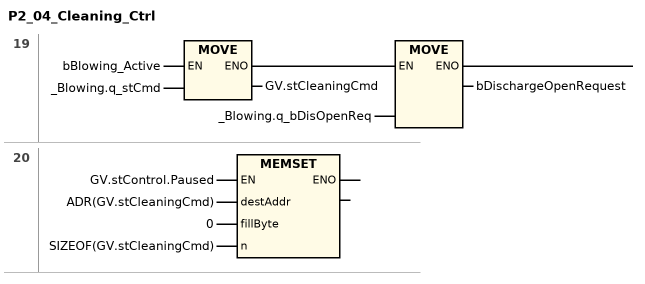
// NETWORK 19
_w4 := bBlowing_Active;
IF _w4 THEN GV.stCleaningCmd := _Blowing.q_stCmd; END_IF
IF _w4 THEN bDischargeOpenRequest := _Blowing.q_bDisOpenReq; END_IF

// NETWORK 20
IF GV.stControl.Paused THEN
    MEMSET(destAddr := ADR(GV.stCleaningCmd), fillByte := 0, n := SIZEOF(GV.stCleaningCmd));
END_IF

END_PROGRAM

// ---- POUs/2. Process/P2_05_Process_Ctrl.TcPOU
PROGRAM P2_05_Process_Ctrl
VAR
	bWaitAferBatchClose			:BOOL;
	tonWaitAfterBatchClose		:TON;
	tonMixerDelayStopped: TON;
END_VAR
VAR // added by the converter: edge detectors and wires of the graphical bodies
    _w1, _w2, _w3 : BOOL;
    _rt1 : R_TRIG;
END_VAR

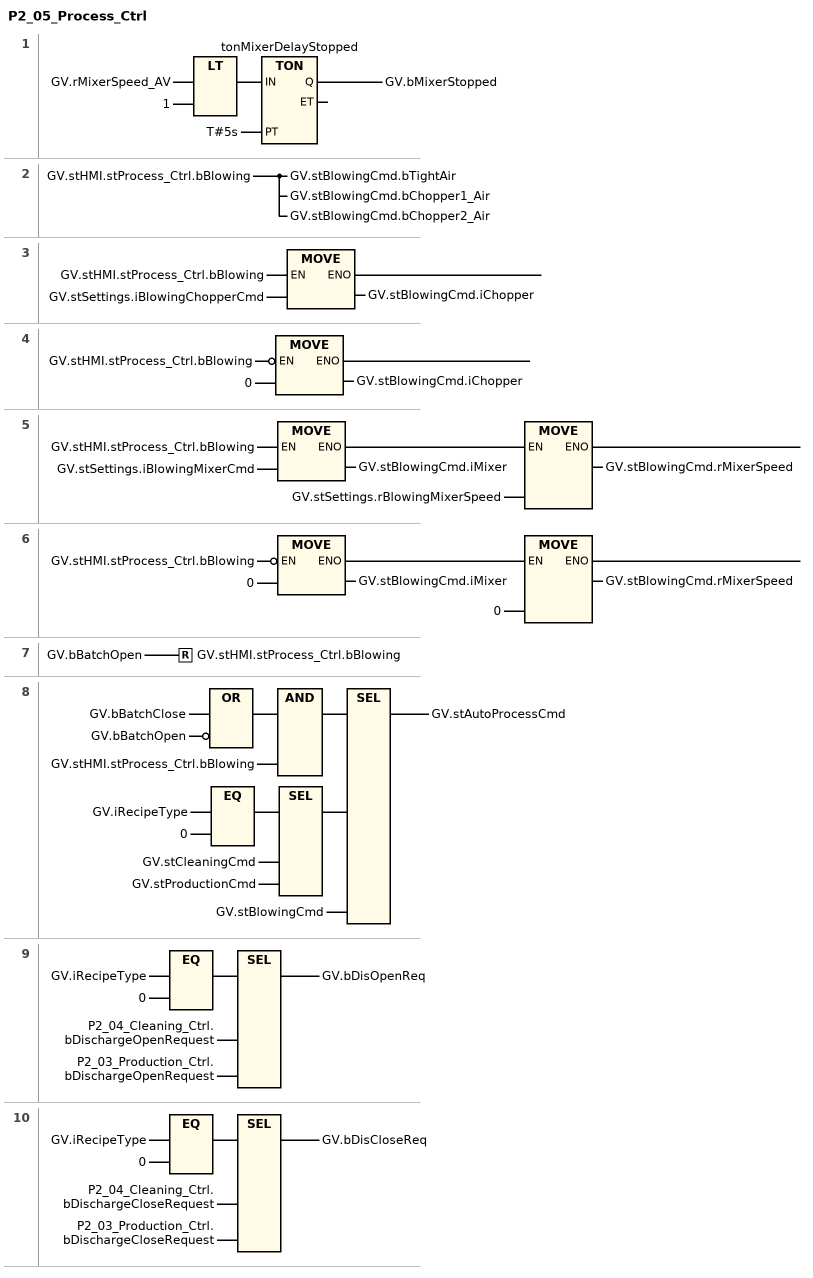
// NETWORK 1
tonMixerDelayStopped(IN := GV.rMixerSpeed_AV < 1, PT := T#5s); // TON
GV.bMixerStopped := tonMixerDelayStopped.Q;

// NETWORK 2
_w1 := GV.stHMI.stProcess_Ctrl.bBlowing;
GV.stBlowingCmd.bTightAir := _w1;
GV.stBlowingCmd.bChopper1_Air := _w1;
GV.stBlowingCmd.bChopper2_Air := _w1;

// NETWORK 3
IF GV.stHMI.stProcess_Ctrl.bBlowing THEN GV.stBlowingCmd.iChopper := GV.stSettings.iBlowingChopperCmd; END_IF

// NETWORK 4
IF NOT GV.stHMI.stProcess_Ctrl.bBlowing THEN GV.stBlowingCmd.iChopper := 0; END_IF

// NETWORK 5
_w2 := GV.stHMI.stProcess_Ctrl.bBlowing;
IF _w2 THEN GV.stBlowingCmd.iMixer := GV.stSettings.iBlowingMixerCmd; END_IF
IF _w2 THEN GV.stBlowingCmd.rMixerSpeed := GV.stSettings.rBlowingMixerSpeed; END_IF

// NETWORK 6
_w3 := NOT GV.stHMI.stProcess_Ctrl.bBlowing;
IF _w3 THEN GV.stBlowingCmd.iMixer := 0; END_IF
IF _w3 THEN GV.stBlowingCmd.rMixerSpeed := 0; END_IF

// NETWORK 7
GV.stHMI.stProcess_Ctrl.bBlowing R= GV.bBatchOpen;

// NETWORK 8
GV.stAutoProcessCmd := SEL((GV.bBatchClose OR NOT GV.bBatchOpen) AND GV.stHMI.stProcess_Ctrl.bBlowing, SEL(GV.iRecipeType = 0, GV.stCleaningCmd, GV.stProductionCmd), GV.stBlowingCmd);

// NETWORK 9
GV.bDisOpenReq := SEL(GV.iRecipeType = 0, P2_04_Cleaning_Ctrl.bDischargeOpenRequest, P2_03_Production_Ctrl.bDischargeOpenRequest);

// NETWORK 10
GV.bDisCloseReq := SEL(GV.iRecipeType = 0, P2_04_Cleaning_Ctrl.bDischargeCloseRequest, P2_03_Production_Ctrl.bDischargeCloseRequest);

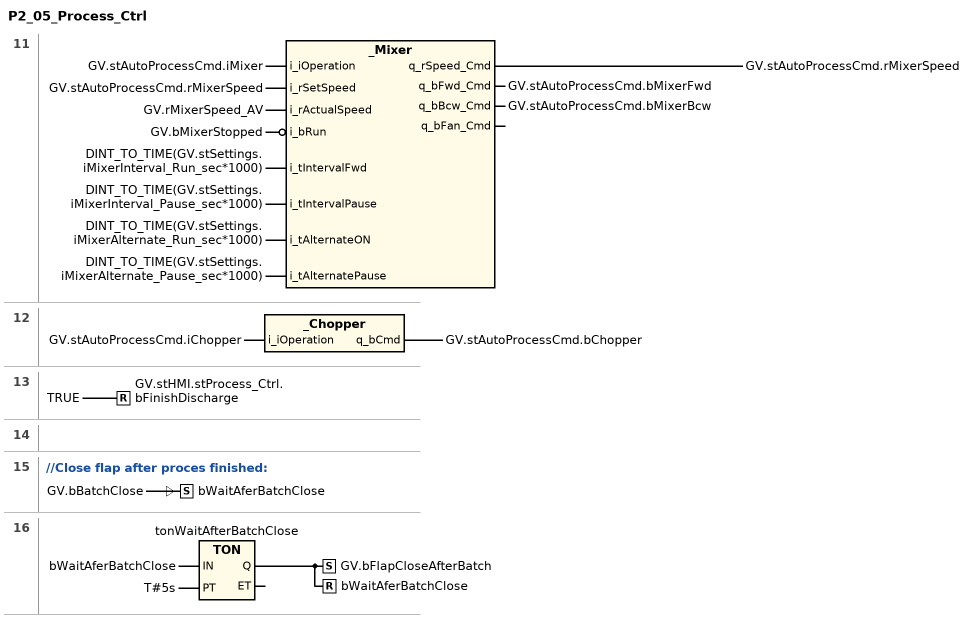
// NETWORK 11
_Mixer(i_iOperation := GV.stAutoProcessCmd.iMixer, i_rSetSpeed := GV.stAutoProcessCmd.rMixerSpeed, i_rActualSpeed := GV.rMixerSpeed_AV, i_bRun := NOT GV.bMixerStopped, i_tIntervalFwd := DINT_TO_TIME(GV.stSettings.iMixerInterval_Run_sec*1000), i_tIntervalPause := DINT_TO_TIME(GV.stSettings.iMixerInterval_Pause_sec*1000), i_tAlternateON := DINT_TO_TIME(GV.stSettings.iMixerAlternate_Run_sec*1000), i_tAlternatePause := DINT_TO_TIME(GV.stSettings.iMixerAlternate_Pause_sec*1000), q_bFwd_Cmd => GV.stAutoProcessCmd.bMixerFwd, q_bBcw_Cmd => GV.stAutoProcessCmd.bMixerBcw);
GV.stAutoProcessCmd.rMixerSpeed := _Mixer.q_rSpeed_Cmd;

// NETWORK 12
_Chopper(i_iOperation := GV.stAutoProcessCmd.iChopper);
GV.stAutoProcessCmd.bChopper := _Chopper.q_bCmd;

// NETWORK 13
GV.stHMI.stProcess_Ctrl.bFinishDischarge R= TRUE;

// NETWORK 14

// NETWORK 15
// label: //Close flap after proces finished
_rt1(CLK := GV.bBatchClose);
bWaitAferBatchClose S= _rt1.Q;

// NETWORK 16
tonWaitAfterBatchClose(IN := bWaitAferBatchClose, PT := T#5s); // TON
GV.bFlapCloseAfterBatch S= tonWaitAfterBatchClose.Q;
bWaitAferBatchClose R= tonWaitAfterBatchClose.Q;

END_PROGRAM

// ---- POUs/2. Process/_Chopper.TcPOU
PROGRAM _Chopper
VAR_INPUT
	i_iOperation			:INT;
END_VAR

VAR
END_VAR

VAR_OUTPUT
	q_bCmd					:BOOL;
END_VAR

IF i_iOperation <> 0 THEN
	IF i_iOperation = 1 THEN
		q_bCmd:=TRUE;
	END_IF
ELSE
	q_bCmd:=FALSE;
END_IF

END_PROGRAM

// ---- POUs/3. Report/P3_00_MAIN.TcPOU
PROGRAM P3_00_MAIN
VAR
	tonDeleteDelay			:TON;
END_VAR

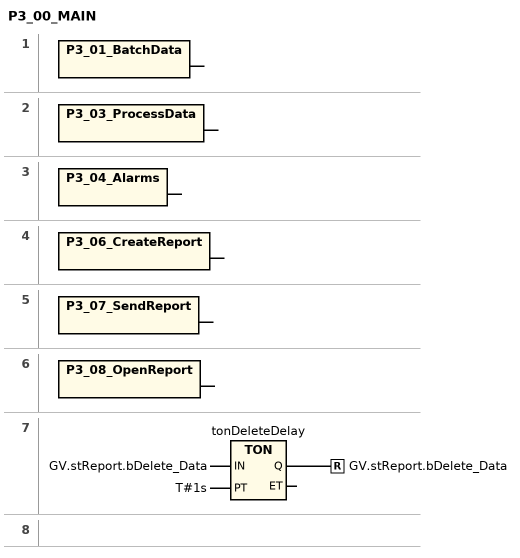
// NETWORK 1
P3_01_BatchData();

// NETWORK 2
P3_03_ProcessData();

// NETWORK 3
P3_04_Alarms();

// NETWORK 4
P3_06_CreateReport();

// NETWORK 5
P3_07_SendReport();

// NETWORK 6
P3_08_OpenReport();

// NETWORK 7
tonDeleteDelay(IN := GV.stReport.bDelete_Data, PT := T#1s); // TON
GV.stReport.bDelete_Data R= tonDeleteDelay.Q;

// NETWORK 8

END_PROGRAM

// ---- POUs/3. Report/P3_01_BatchData.TcPOU
PROGRAM P3_01_BatchData
VAR
	
	arrBatchParam				:ARRAY[0..19] OF STRING;
	arrBatchValue				:ARRAY[0..19] OF STRING;
	
	iNoParameters				:INT;
	
	stDBParam 					:ST_BatchData;	
	fbDBWrite					:FB_PLCDBWriteEvt(sNetId:=CONST.AMS_NETID, tTimeout:=DEFAULT_ADS_TIMEOUT);
	tableColumns				:ARRAY [0..2] OF STRING(50) := ['Batch', 'Parameter', 'Value'];
	arrParam					:ARRAY [0..2] OF ST_ExpParameter := [(sParaName := 'Batch', nParaSize := 101, eParaType := E_EXPPARAMETERTYPE.STRING_), 
																	(sParaName := 'Parameter', nParaSize := 101, eParaType := E_EXPPARAMETERTYPE.STRING_),
															 		(sParaName := 'Value', nParaSize := 101, eParaType := E_EXPPARAMETERTYPE.STRING_)];
															 
	fbDeleteTable    			:FB_PLCDBCmdEvt(sNetID:=CONST.AMS_NETID, tTimeout:=DEFAULT_ADS_TIMEOUT);	
	sDelete						:STRING;	
	bDelete						:BOOL;
															 
	bWrite						:BOOL;
	iWrite						:USINT;
	bStartWrite					:BOOL;
	
	sVersion					:STRING;
	
	iStepWrite					:INT;
	trigStartWrite				:R_TRIG;
	tonDelayWrite				:TON;
	
END_VAR
VAR PERSISTENT
	dtBatchOpen					:DT;
	dtBatchClose				:DT;
	
	ulBatchOpen					:ULINT;
	ulBatchClose				:ULINT;
END_VAR
VAR // added by the converter: edge detectors and wires of the graphical bodies
    _rt1, _rt2 : R_TRIG;
    _w1, _w2 : BOOL;
END_VAR

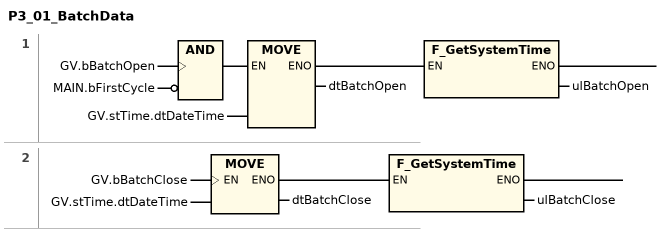
// NETWORK 1
_rt1(CLK := GV.bBatchOpen);
_w1 := _rt1.Q AND NOT MAIN.bFirstCycle;
IF _w1 THEN dtBatchOpen := GV.stTime.dtDateTime; END_IF
IF _w1 THEN ulBatchOpen := F_GetSystemTime(); END_IF

// NETWORK 2
_rt2(CLK := GV.bBatchClose);
_w2 := _rt2.Q;
IF _w2 THEN dtBatchClose := GV.stTime.dtDateTime; END_IF
IF _w2 THEN ulBatchClose := F_GetSystemTime(); END_IF

END_PROGRAM

// ---- POUs/3. Report/P3_03_ProcessData.TcPOU
PROGRAM P3_03_ProcessData
VAR
	stDBParam 					:ST_ProcessData;	

	fbDBWrite					:FB_PLCDBWriteEvt(sNetId:=CONST.AMS_NETID, tTimeout:=DEFAULT_ADS_TIMEOUT);
	tableColumns				:ARRAY [0..8] OF STRING(50) := ['Batch', 'DateTime', 'Value1', 'Value2', 'Value3', 'Value4', 'Value5', 'Value6', 'Value7'];
	arrParam					:ARRAY [0..8] OF ST_ExpParameter := [(sParaName := 'Batch', nParaSize := 101, eParaType := E_EXPPARAMETERTYPE.STRING_),
															 (sParaName := 'DateTime', nParaSize := 4, eParaType := E_EXPPARAMETERTYPE.DateTime), 
															 (sParaName := 'Value1', nParaSize := 101, eParaType := E_EXPPARAMETERTYPE.STRING_), 
															 (sParaName := 'Value2', nParaSize := 101, eParaType := E_EXPPARAMETERTYPE.STRING_), 
															 (sParaName := 'Value3', nParaSize := 101, eParaType := E_EXPPARAMETERTYPE.STRING_),
															 (sParaName := 'Value4', nParaSize := 101, eParaType := E_EXPPARAMETERTYPE.STRING_),
															 (sParaName := 'Value5', nParaSize := 101, eParaType := E_EXPPARAMETERTYPE.STRING_),
															 (sParaName := 'Value6', nParaSize := 101, eParaType := E_EXPPARAMETERTYPE.STRING_),
															 (sParaName := 'Value7', nParaSize := 101, eParaType := E_EXPPARAMETERTYPE.STRING_)];
		
	fbDeleteTable    			:FB_PLCDBCmdEvt(sNetID:=CONST.AMS_NETID, tTimeout:=DEFAULT_ADS_TIMEOUT);	
	sDelete						:STRING;	
	bDelete						:BOOL;
										 
	bWrite						:BOOL;	
	
	sChopper1Speed				:STRING;
	sChopper2Speed				:STRING;
END_VAR
VAR // added by the converter: edge detectors and wires of the graphical bodies
    _rt1, _rt2 : R_TRIG;
END_VAR

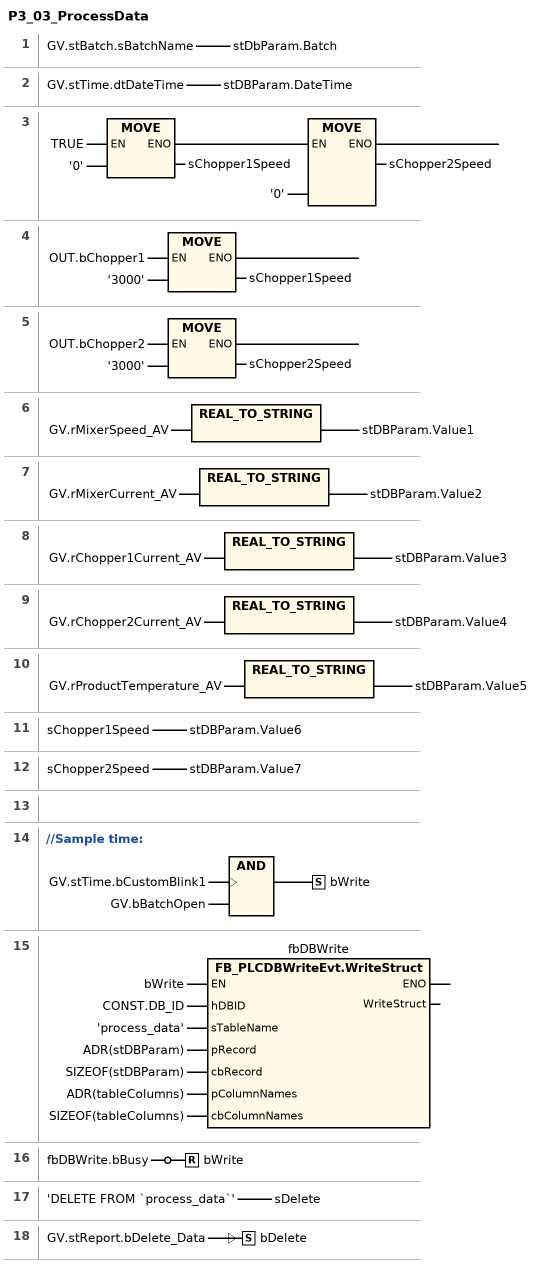
// NETWORK 1
stDbParam.Batch := GV.stBatch.sBatchName;

// NETWORK 2
stDBParam.DateTime := GV.stTime.dtDateTime;

// NETWORK 3
sChopper1Speed := '0';
sChopper2Speed := '0';

// NETWORK 4
IF OUT.bChopper1 THEN sChopper1Speed := '3000'; END_IF

// NETWORK 5
IF OUT.bChopper2 THEN sChopper2Speed := '3000'; END_IF

// NETWORK 6
stDBParam.Value1 := REAL_TO_STRING(GV.rMixerSpeed_AV);

// NETWORK 7
stDBParam.Value2 := REAL_TO_STRING(GV.rMixerCurrent_AV);

// NETWORK 8
stDBParam.Value3 := REAL_TO_STRING(GV.rChopper1Current_AV);

// NETWORK 9
stDBParam.Value4 := REAL_TO_STRING(GV.rChopper2Current_AV);

// NETWORK 10
stDBParam.Value5 := REAL_TO_STRING(GV.rProductTemperature_AV);

// NETWORK 11
stDBParam.Value6 := sChopper1Speed;

// NETWORK 12
stDBParam.Value7 := sChopper2Speed;

// NETWORK 13

// NETWORK 14
// label: //Sample time
_rt1(CLK := GV.stTime.bCustomBlink1);
bWrite S= _rt1.Q AND GV.bBatchOpen;

// NETWORK 15
IF bWrite THEN
    fbDBWrite.WriteStruct(
        hDBID := CONST.DB_ID,
        sTableName := 'process_data',
        pRecord := ADR(stDBParam),
        cbRecord := SIZEOF(stDBParam),
        pColumnNames := ADR(tableColumns),
        cbColumnNames := SIZEOF(tableColumns));
END_IF

// NETWORK 16
bWrite R= NOT fbDBWrite.bBusy;

// NETWORK 17
sDelete := 'DELETE FROM `process_data`';

// NETWORK 18
_rt2(CLK := GV.stReport.bDelete_Data);
bDelete S= _rt2.Q;

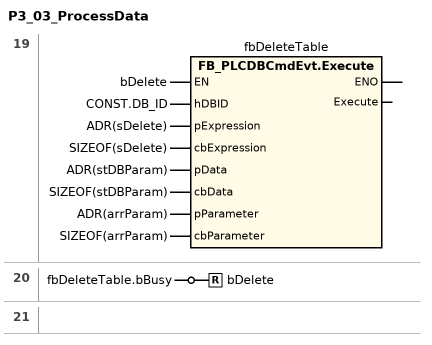
// NETWORK 19
IF bDelete THEN
    fbDeleteTable.Execute(
        hDBID := CONST.DB_ID,
        pExpression := ADR(sDelete),
        cbExpression := SIZEOF(sDelete),
        pData := ADR(stDBParam),
        cbData := SIZEOF(stDBParam),
        pParameter := ADR(arrParam),
        cbParameter := SIZEOF(arrParam));
END_IF

// NETWORK 20
bDelete R= NOT fbDeleteTable.bBusy;

// NETWORK 21

END_PROGRAM

// ---- POUs/3. Report/P3_04_Alarms.TcPOU
PROGRAM P3_04_Alarms
VAR 
	fbEventLogger		:FB_TcEventLogger;
	fbCsvExportSetting	:FB_TcEventCsvExportSettings;
	fbExportFilter		:FB_TcEventFilter;

	fbTrig				:R_TRIG;
	
	ulFilter1			:ULINT;
	ulFilter2			:ULINT;
	
	sPath				:STRING;
	
	
END_VAR

//Link here...

ulFilter1:=P3_01_BatchData.ulBatchOpen;
ulFilter2:=P3_01_BatchData.ulBatchClose;

fbTrig(CLK:=GV.stReport.bExport_Alarms);
IF GV.stReport.bExport_Alarms THEN
	IF fbTrig.Q THEN
		fbCsvExportSetting.Clear();
		fbCsvExportSetting.bWithHeader:=TRUE;
		fbCsvExportSetting.sDelimiter:=',';
		fbCsvExportSetting.AddFilter(fbExportFilter);
		fbExportFilter.Clear();
		fbExportFilter.IsAlarm().AND_OP().
		TimeRaised.GreaterThanOrEqualTo(ulFilter1).AND_OP().
		TimeRaised.LessThanOrEqualTo(ulFilter2).AND_OP().
		Source.Name.EqualTo('GV.stAlarm');
	END_IF
	
	sPath:=CONCAT(CONST.PROJECT_DIR,'Reports\1. Raw Data\AlarmLog.txt');
	
	IF fbEventLogger.ExportLoggedEvents(sPath,fbCsvExportSetting) THEN
		GV.stReport.bExport_Alarms:=FALSE;
	END_IF
END_IF

END_PROGRAM

// ---- POUs/3. Report/P3_08_OpenReport.TcPOU
PROGRAM P3_08_OpenReport
VAR
	sDateTime			:STRING;
	sYear				:STRING;
	sMonth				:STRING;
	sDay				:STRING;
	sHour				:STRING;
	sMinute				:STRING;
	sReportSuffix		:STRING;
END_VAR

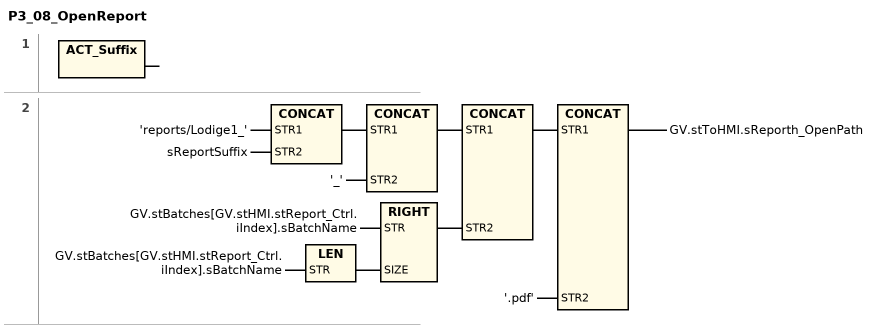
// NETWORK 1
ACT_Suffix();

// NETWORK 2
GV.stToHMI.sReporth_OpenPath := CONCAT(STR1 := CONCAT(STR1 := CONCAT(STR1 := CONCAT(STR1 := 'reports/Lodige1_', STR2 := sReportSuffix), STR2 := '_'), STR2 := RIGHT(STR := GV.stBatches[GV.stHMI.stReport_Ctrl.iIndex].sBatchName, SIZE := LEN(STR := GV.stBatches[GV.stHMI.stReport_Ctrl.iIndex].sBatchName))), STR2 := '.pdf');

ACTION ACT_Suffix:
sDateTime:=GV.stBatches[GV.stHMI.stReport_Ctrl.iIndex].sFinished;
sYear:=RIGHT(LEFT(sDateTime,10),2);
sMonth:=RIGHT(LEFT(sDateTime,5),2);
sDay:=LEFT(sDateTime,2);

sHour:=LEFT(RIGHT(sDateTime,8),2);
sMinute:=LEFT(RIGHT(sDateTime,5),2);

sReportSuffix:=CONCAT(sYear,sMonth);
sReportSuffix:=CONCAT(sReportSuffix,sDay);
sReportSuffix:=CONCAT(sReportSuffix,sHour);
sReportSuffix:=CONCAT(sReportSuffix,sMinute);
END_ACTION

END_PROGRAM

// ---- POUs/4. Audit Trail/P4_00_MAIN.TcPOU
PROGRAM P4_00_MAIN
VAR
END_VAR

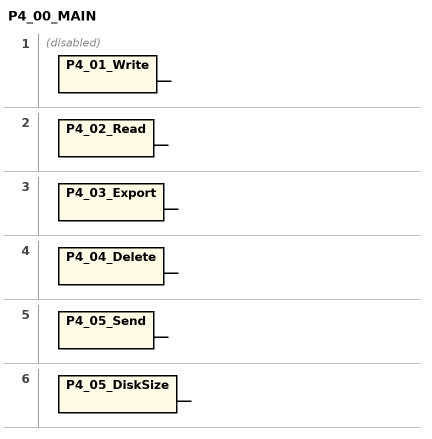
// NETWORK 1 (disabled)
// P4_01_Write();

// NETWORK 2
P4_02_Read();

// NETWORK 3
P4_03_Export();

// NETWORK 4
P4_04_Delete();

// NETWORK 5
P4_05_Send();

// NETWORK 6
P4_05_DiskSize();

END_PROGRAM

// ---- POUs/4. Audit Trail/P4_01_Write.TcPOU
PROGRAM P4_01_Write
VAR
	stDBParam 				:ST_AuditTrail;	
	tableColumns			:ARRAY [0..5] OF STRING(50) := ['DateTime', 'User', 'Event', 'Description', 'OldValue', 'NewValue'];	

	fbDBWrite				:FB_PLCDBWriteEvt(sNetId:=CONST.AMS_NETID, tTimeout:=DEFAULT_ADS_TIMEOUT);	
	bWrite					:BOOL;
	

	
	fbRecipeProdValue		:ARRAY[0..9] OF FB_WriteChange;
	fbRecipeProdStrings		:ARRAY[0..9] OF FB_WriteChange_STR;
	fbRecipeProdClick		:ARRAY[0..9] OF FB_WriteClick;
	bRecipeProdChange		:ARRAY[0..19] OF BOOL;
	
	fbRecipeCleanValue		:ARRAY[0..29] OF FB_WriteChange;
	fbRecipeCleanStrings	:ARRAY[0..29] OF FB_WriteChange_STR;
	fbRecipeCleanClick		:ARRAY[0..29] OF FB_WriteClick;
	bRecipeCleanChange		:ARRAY[0..39] OF BOOL;
	
	fbBatchProdValue		:ARRAY[0..9] OF FB_WriteChange;
	fbBatchProdStrings		:ARRAY[0..9] OF FB_WriteChange_STR;
	fbBatchProdClick		:ARRAY[0..9] OF FB_WriteClick;
	bBatchProdChange		:ARRAY[0..19] OF BOOL;
	
	fbBatchCleanValue		:ARRAY[0..29] OF FB_WriteChange;
	fbBatchCleanStrings		:ARRAY[0..29] OF FB_WriteChange_STR;
	fbBatchCleanClick		:ARRAY[0..29] OF FB_WriteClick;
	bBatchCleanChange		:ARRAY[0..39] OF BOOL;
	
	
	fbSettingsChange		:ARRAY[0..19] OF FB_WriteChange;
	bSettingsChange			:ARRAY[0..19] OF BOOL;	
	
	fbAlarmsettChange		:ARRAY[0..9] OF FB_WriteChange;
	bAlarmsettChange		:ARRAY[0..9] OF BOOL;
	
	fbOperatorAction		:ARRAY[0..39] OF FB_WriteClick;
	bOperatorAction			:ARRAY[0..39] OF BOOL;

	bScanBatchParams		:BOOL;
	
END_VAR
VAR // added by the converter: edge detectors and wires of the graphical bodies
    _rt1 : R_TRIG;
END_VAR

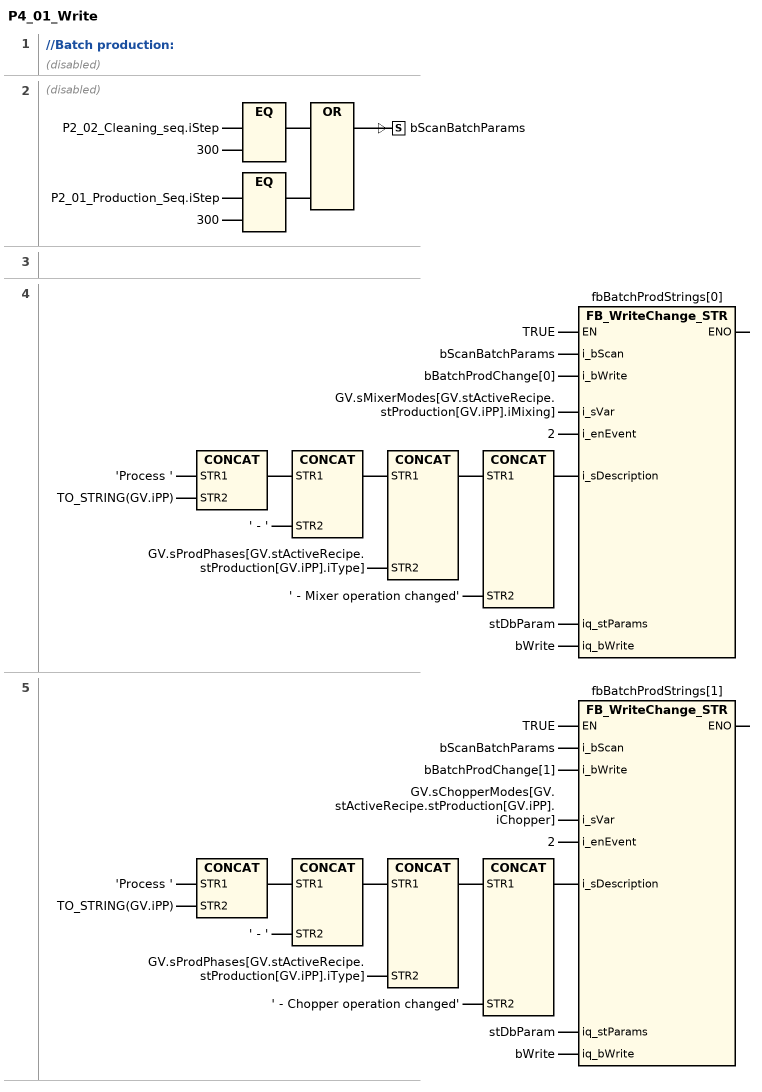
// NETWORK 1 (disabled)
// label: //Batch production

// NETWORK 2 (disabled)
// _rt1(CLK := P2_02_Cleaning_seq.iStep = 300 OR P2_01_Production_Seq.iStep = 300);
// bScanBatchParams S= _rt1.Q;

// NETWORK 3

// NETWORK 4
fbBatchProdStrings[0](
    i_bScan := bScanBatchParams,
    i_bWrite := bBatchProdChange[0],
    i_sVar := GV.sMixerModes[GV.stActiveRecipe.stProduction[GV.iPP].iMixing],
    i_enEvent := 2,
    i_sDescription := CONCAT(STR1 := CONCAT(STR1 := CONCAT(STR1 := CONCAT(STR1 := 'Process ', STR2 := TO_STRING(GV.iPP)), STR2 := ' - '), STR2 := GV.sProdPhases[GV.stActiveRecipe.stProduction[GV.iPP].iType]), STR2 := ' - Mixer operation changed'),
    iq_stParams := stDbParam,
    iq_bWrite := bWrite); // FB_WriteChange_STR

// NETWORK 5
fbBatchProdStrings[1](
    i_bScan := bScanBatchParams,
    i_bWrite := bBatchProdChange[1],
    i_sVar := GV.sChopperModes[GV.stActiveRecipe.stProduction[GV.iPP].iChopper],
    i_enEvent := 2,
    i_sDescription := CONCAT(STR1 := CONCAT(STR1 := CONCAT(STR1 := CONCAT(STR1 := 'Process ', STR2 := TO_STRING(GV.iPP)), STR2 := ' - '), STR2 := GV.sProdPhases[GV.stActiveRecipe.stProduction[GV.iPP].iType]), STR2 := ' - Chopper operation changed'),
    iq_stParams := stDbParam,
    iq_bWrite := bWrite); // FB_WriteChange_STR

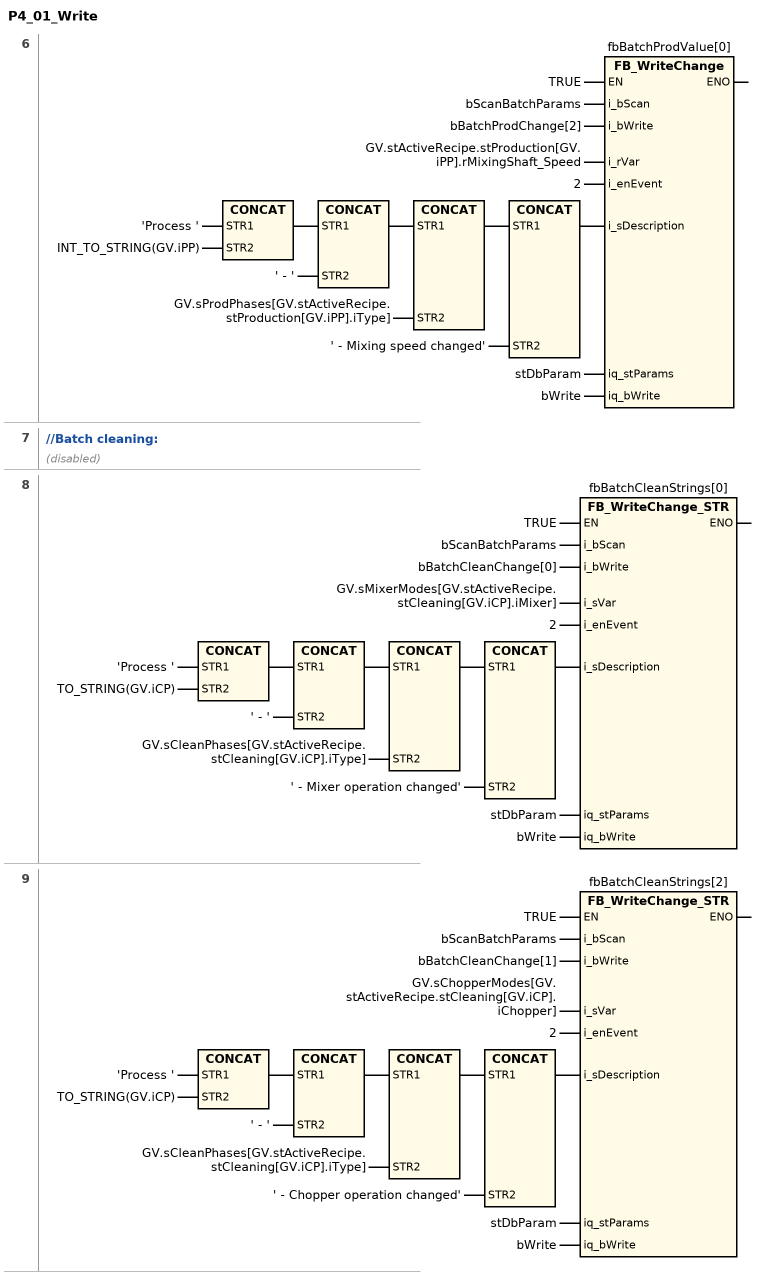
// NETWORK 6
fbBatchProdValue[0](
    i_bScan := bScanBatchParams,
    i_bWrite := bBatchProdChange[2],
    i_rVar := GV.stActiveRecipe.stProduction[GV.iPP].rMixingShaft_Speed,
    i_enEvent := 2,
    i_sDescription := CONCAT(STR1 := CONCAT(STR1 := CONCAT(STR1 := CONCAT(STR1 := 'Process ', STR2 := INT_TO_STRING(GV.iPP)), STR2 := ' - '), STR2 := GV.sProdPhases[GV.stActiveRecipe.stProduction[GV.iPP].iType]), STR2 := ' - Mixing speed changed'),
    iq_stParams := stDbParam,
    iq_bWrite := bWrite); // FB_WriteChange

// NETWORK 7 (disabled)
// label: //Batch cleaning

// NETWORK 8
fbBatchCleanStrings[0](
    i_bScan := bScanBatchParams,
    i_bWrite := bBatchCleanChange[0],
    i_sVar := GV.sMixerModes[GV.stActiveRecipe.stCleaning[GV.iCP].iMixer],
    i_enEvent := 2,
    i_sDescription := CONCAT(STR1 := CONCAT(STR1 := CONCAT(STR1 := CONCAT(STR1 := 'Process ', STR2 := TO_STRING(GV.iCP)), STR2 := ' - '), STR2 := GV.sCleanPhases[GV.stActiveRecipe.stCleaning[GV.iCP].iType]), STR2 := ' - Mixer operation changed'),
    iq_stParams := stDbParam,
    iq_bWrite := bWrite); // FB_WriteChange_STR

// NETWORK 9
fbBatchCleanStrings[2](
    i_bScan := bScanBatchParams,
    i_bWrite := bBatchCleanChange[1],
    i_sVar := GV.sChopperModes[GV.stActiveRecipe.stCleaning[GV.iCP].iChopper],
    i_enEvent := 2,
    i_sDescription := CONCAT(STR1 := CONCAT(STR1 := CONCAT(STR1 := CONCAT(STR1 := 'Process ', STR2 := TO_STRING(GV.iCP)), STR2 := ' - '), STR2 := GV.sCleanPhases[GV.stActiveRecipe.stCleaning[GV.iCP].iType]), STR2 := ' - Chopper operation changed'),
    iq_stParams := stDbParam,
    iq_bWrite := bWrite); // FB_WriteChange_STR

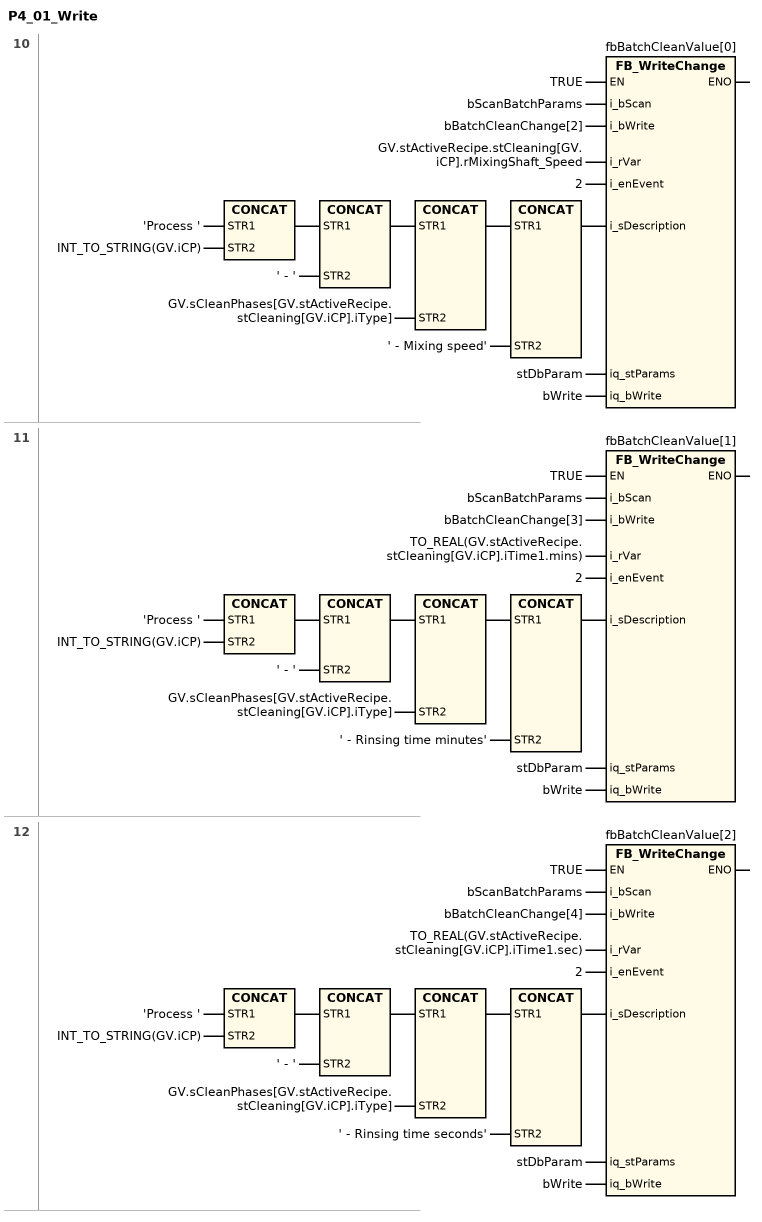
// NETWORK 10
fbBatchCleanValue[0](
    i_bScan := bScanBatchParams,
    i_bWrite := bBatchCleanChange[2],
    i_rVar := GV.stActiveRecipe.stCleaning[GV.iCP].rMixingShaft_Speed,
    i_enEvent := 2,
    i_sDescription := CONCAT(STR1 := CONCAT(STR1 := CONCAT(STR1 := CONCAT(STR1 := 'Process ', STR2 := INT_TO_STRING(GV.iCP)), STR2 := ' - '), STR2 := GV.sCleanPhases[GV.stActiveRecipe.stCleaning[GV.iCP].iType]), STR2 := ' - Mixing speed'),
    iq_stParams := stDbParam,
    iq_bWrite := bWrite); // FB_WriteChange

// NETWORK 11
fbBatchCleanValue[1](
    i_bScan := bScanBatchParams,
    i_bWrite := bBatchCleanChange[3],
    i_rVar := TO_REAL(GV.stActiveRecipe.stCleaning[GV.iCP].iTime1.mins),
    i_enEvent := 2,
    i_sDescription := CONCAT(STR1 := CONCAT(STR1 := CONCAT(STR1 := CONCAT(STR1 := 'Process ', STR2 := INT_TO_STRING(GV.iCP)), STR2 := ' - '), STR2 := GV.sCleanPhases[GV.stActiveRecipe.stCleaning[GV.iCP].iType]), STR2 := ' - Rinsing time minutes'),
    iq_stParams := stDbParam,
    iq_bWrite := bWrite); // FB_WriteChange

// NETWORK 12
fbBatchCleanValue[2](
    i_bScan := bScanBatchParams,
    i_bWrite := bBatchCleanChange[4],
    i_rVar := TO_REAL(GV.stActiveRecipe.stCleaning[GV.iCP].iTime1.sec),
    i_enEvent := 2,
    i_sDescription := CONCAT(STR1 := CONCAT(STR1 := CONCAT(STR1 := CONCAT(STR1 := 'Process ', STR2 := INT_TO_STRING(GV.iCP)), STR2 := ' - '), STR2 := GV.sCleanPhases[GV.stActiveRecipe.stCleaning[GV.iCP].iType]), STR2 := ' - Rinsing time seconds'),
    iq_stParams := stDbParam,
    iq_bWrite := bWrite); // FB_WriteChange

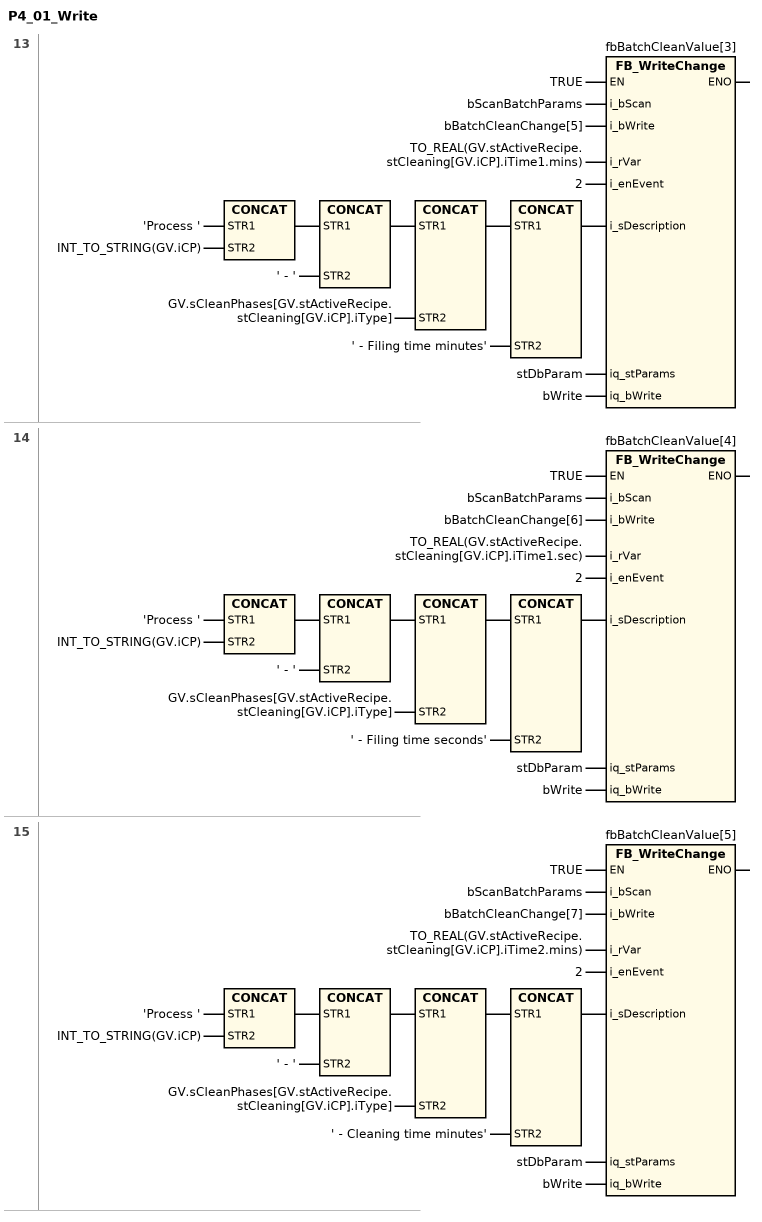
// NETWORK 13
fbBatchCleanValue[3](
    i_bScan := bScanBatchParams,
    i_bWrite := bBatchCleanChange[5],
    i_rVar := TO_REAL(GV.stActiveRecipe.stCleaning[GV.iCP].iTime1.mins),
    i_enEvent := 2,
    i_sDescription := CONCAT(STR1 := CONCAT(STR1 := CONCAT(STR1 := CONCAT(STR1 := 'Process ', STR2 := INT_TO_STRING(GV.iCP)), STR2 := ' - '), STR2 := GV.sCleanPhases[GV.stActiveRecipe.stCleaning[GV.iCP].iType]), STR2 := ' - Filing time minutes'),
    iq_stParams := stDbParam,
    iq_bWrite := bWrite); // FB_WriteChange

// NETWORK 14
fbBatchCleanValue[4](
    i_bScan := bScanBatchParams,
    i_bWrite := bBatchCleanChange[6],
    i_rVar := TO_REAL(GV.stActiveRecipe.stCleaning[GV.iCP].iTime1.sec),
    i_enEvent := 2,
    i_sDescription := CONCAT(STR1 := CONCAT(STR1 := CONCAT(STR1 := CONCAT(STR1 := 'Process ', STR2 := INT_TO_STRING(GV.iCP)), STR2 := ' - '), STR2 := GV.sCleanPhases[GV.stActiveRecipe.stCleaning[GV.iCP].iType]), STR2 := ' - Filing time seconds'),
    iq_stParams := stDbParam,
    iq_bWrite := bWrite); // FB_WriteChange

// NETWORK 15
fbBatchCleanValue[5](
    i_bScan := bScanBatchParams,
    i_bWrite := bBatchCleanChange[7],
    i_rVar := TO_REAL(GV.stActiveRecipe.stCleaning[GV.iCP].iTime2.mins),
    i_enEvent := 2,
    i_sDescription := CONCAT(STR1 := CONCAT(STR1 := CONCAT(STR1 := CONCAT(STR1 := 'Process ', STR2 := INT_TO_STRING(GV.iCP)), STR2 := ' - '), STR2 := GV.sCleanPhases[GV.stActiveRecipe.stCleaning[GV.iCP].iType]), STR2 := ' - Cleaning time minutes'),
    iq_stParams := stDbParam,
    iq_bWrite := bWrite); // FB_WriteChange

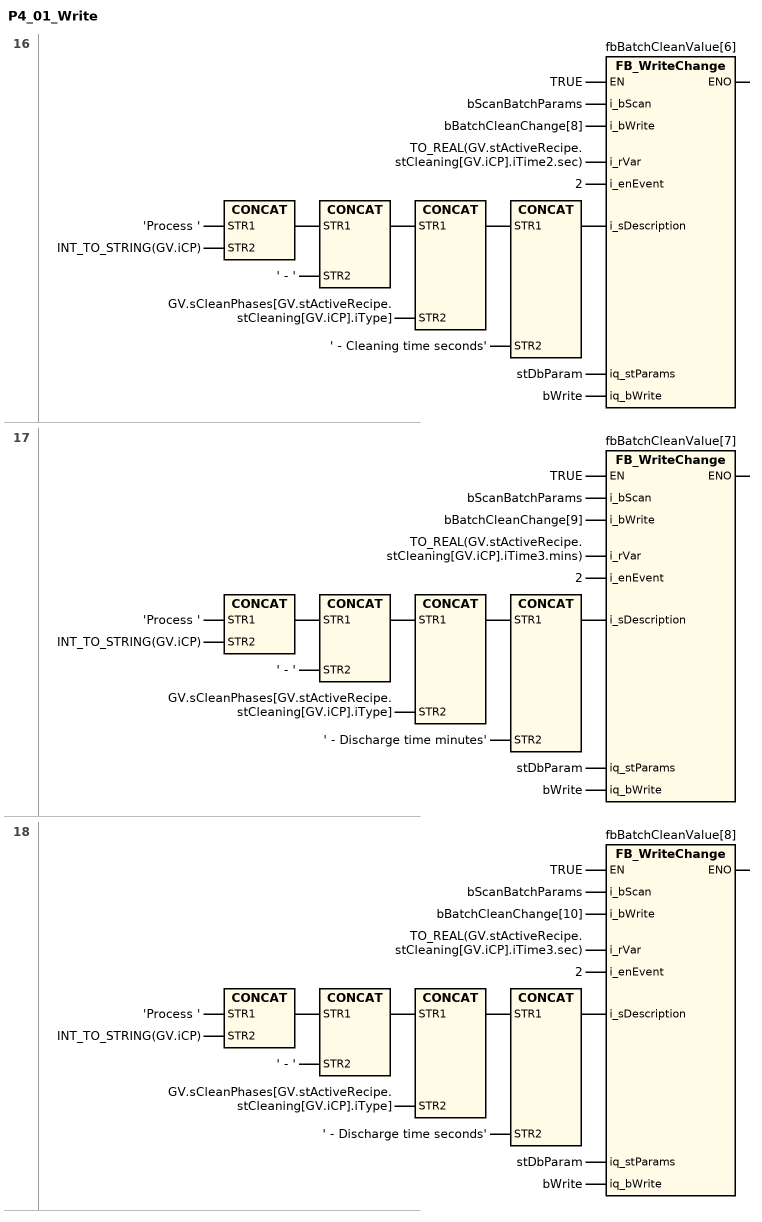
// NETWORK 16
fbBatchCleanValue[6](
    i_bScan := bScanBatchParams,
    i_bWrite := bBatchCleanChange[8],
    i_rVar := TO_REAL(GV.stActiveRecipe.stCleaning[GV.iCP].iTime2.sec),
    i_enEvent := 2,
    i_sDescription := CONCAT(STR1 := CONCAT(STR1 := CONCAT(STR1 := CONCAT(STR1 := 'Process ', STR2 := INT_TO_STRING(GV.iCP)), STR2 := ' - '), STR2 := GV.sCleanPhases[GV.stActiveRecipe.stCleaning[GV.iCP].iType]), STR2 := ' - Cleaning time seconds'),
    iq_stParams := stDbParam,
    iq_bWrite := bWrite); // FB_WriteChange

// NETWORK 17
fbBatchCleanValue[7](
    i_bScan := bScanBatchParams,
    i_bWrite := bBatchCleanChange[9],
    i_rVar := TO_REAL(GV.stActiveRecipe.stCleaning[GV.iCP].iTime3.mins),
    i_enEvent := 2,
    i_sDescription := CONCAT(STR1 := CONCAT(STR1 := CONCAT(STR1 := CONCAT(STR1 := 'Process ', STR2 := INT_TO_STRING(GV.iCP)), STR2 := ' - '), STR2 := GV.sCleanPhases[GV.stActiveRecipe.stCleaning[GV.iCP].iType]), STR2 := ' - Discharge time minutes'),
    iq_stParams := stDbParam,
    iq_bWrite := bWrite); // FB_WriteChange

// NETWORK 18
fbBatchCleanValue[8](
    i_bScan := bScanBatchParams,
    i_bWrite := bBatchCleanChange[10],
    i_rVar := TO_REAL(GV.stActiveRecipe.stCleaning[GV.iCP].iTime3.sec),
    i_enEvent := 2,
    i_sDescription := CONCAT(STR1 := CONCAT(STR1 := CONCAT(STR1 := CONCAT(STR1 := 'Process ', STR2 := INT_TO_STRING(GV.iCP)), STR2 := ' - '), STR2 := GV.sCleanPhases[GV.stActiveRecipe.stCleaning[GV.iCP].iType]), STR2 := ' - Discharge time seconds'),
    iq_stParams := stDbParam,
    iq_bWrite := bWrite); // FB_WriteChange

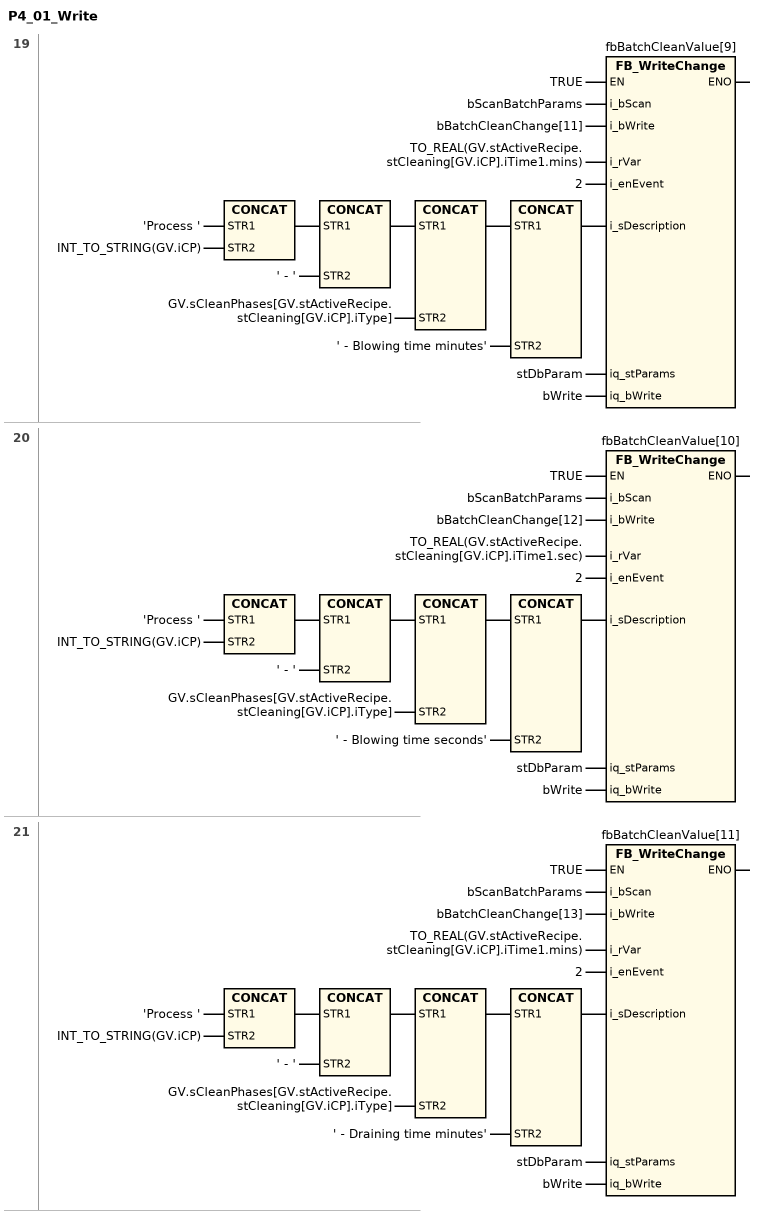
// NETWORK 19
fbBatchCleanValue[9](
    i_bScan := bScanBatchParams,
    i_bWrite := bBatchCleanChange[11],
    i_rVar := TO_REAL(GV.stActiveRecipe.stCleaning[GV.iCP].iTime1.mins),
    i_enEvent := 2,
    i_sDescription := CONCAT(STR1 := CONCAT(STR1 := CONCAT(STR1 := CONCAT(STR1 := 'Process ', STR2 := INT_TO_STRING(GV.iCP)), STR2 := ' - '), STR2 := GV.sCleanPhases[GV.stActiveRecipe.stCleaning[GV.iCP].iType]), STR2 := ' - Blowing time minutes'),
    iq_stParams := stDbParam,
    iq_bWrite := bWrite); // FB_WriteChange

// NETWORK 20
fbBatchCleanValue[10](
    i_bScan := bScanBatchParams,
    i_bWrite := bBatchCleanChange[12],
    i_rVar := TO_REAL(GV.stActiveRecipe.stCleaning[GV.iCP].iTime1.sec),
    i_enEvent := 2,
    i_sDescription := CONCAT(STR1 := CONCAT(STR1 := CONCAT(STR1 := CONCAT(STR1 := 'Process ', STR2 := INT_TO_STRING(GV.iCP)), STR2 := ' - '), STR2 := GV.sCleanPhases[GV.stActiveRecipe.stCleaning[GV.iCP].iType]), STR2 := ' - Blowing time seconds'),
    iq_stParams := stDbParam,
    iq_bWrite := bWrite); // FB_WriteChange

// NETWORK 21
fbBatchCleanValue[11](
    i_bScan := bScanBatchParams,
    i_bWrite := bBatchCleanChange[13],
    i_rVar := TO_REAL(GV.stActiveRecipe.stCleaning[GV.iCP].iTime1.mins),
    i_enEvent := 2,
    i_sDescription := CONCAT(STR1 := CONCAT(STR1 := CONCAT(STR1 := CONCAT(STR1 := 'Process ', STR2 := INT_TO_STRING(GV.iCP)), STR2 := ' - '), STR2 := GV.sCleanPhases[GV.stActiveRecipe.stCleaning[GV.iCP].iType]), STR2 := ' - Draining time minutes'),
    iq_stParams := stDbParam,
    iq_bWrite := bWrite); // FB_WriteChange

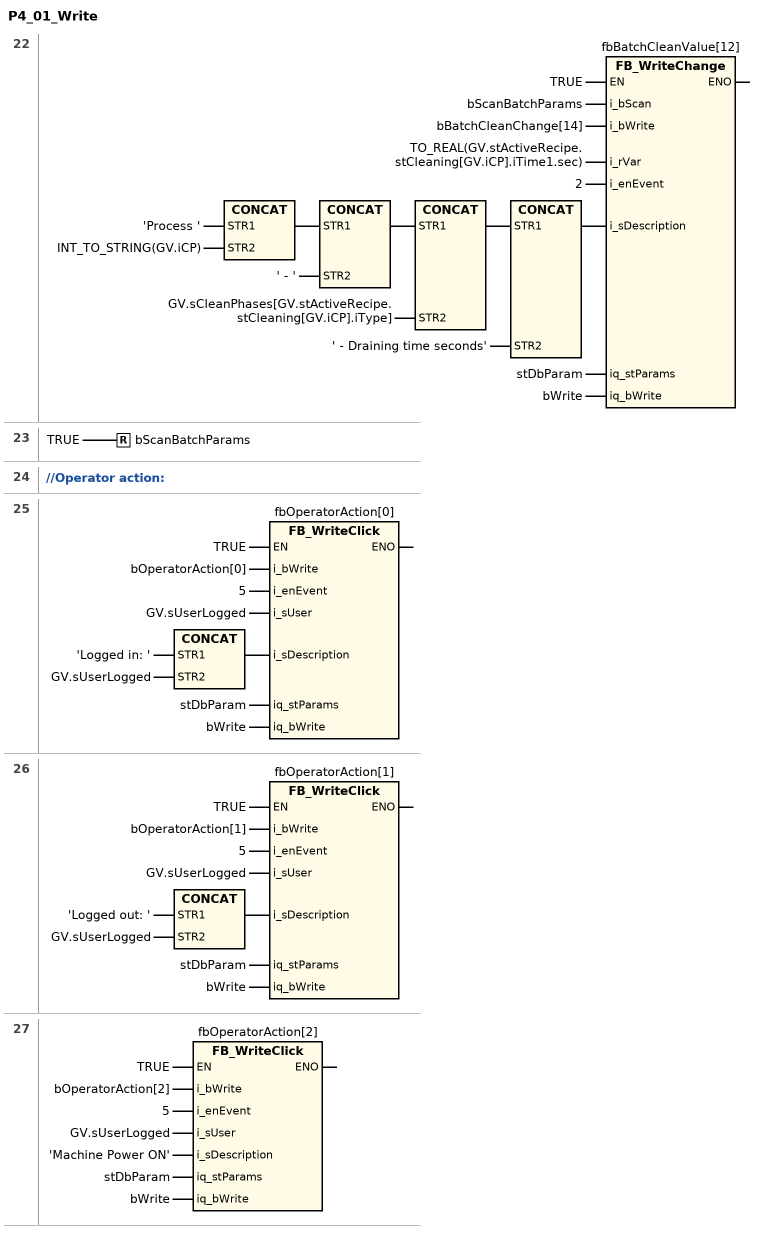
// NETWORK 22
fbBatchCleanValue[12](
    i_bScan := bScanBatchParams,
    i_bWrite := bBatchCleanChange[14],
    i_rVar := TO_REAL(GV.stActiveRecipe.stCleaning[GV.iCP].iTime1.sec),
    i_enEvent := 2,
    i_sDescription := CONCAT(STR1 := CONCAT(STR1 := CONCAT(STR1 := CONCAT(STR1 := 'Process ', STR2 := INT_TO_STRING(GV.iCP)), STR2 := ' - '), STR2 := GV.sCleanPhases[GV.stActiveRecipe.stCleaning[GV.iCP].iType]), STR2 := ' - Draining time seconds'),
    iq_stParams := stDbParam,
    iq_bWrite := bWrite); // FB_WriteChange

// NETWORK 23
bScanBatchParams R= TRUE;

// NETWORK 24
// label: //Operator action

// NETWORK 25
fbOperatorAction[0](
    i_bWrite := bOperatorAction[0],
    i_enEvent := 5,
    i_sUser := GV.sUserLogged,
    i_sDescription := CONCAT(STR1 := 'Logged in: ', STR2 := GV.sUserLogged),
    iq_stParams := stDbParam,
    iq_bWrite := bWrite); // FB_WriteClick

// NETWORK 26
fbOperatorAction[1](
    i_bWrite := bOperatorAction[1],
    i_enEvent := 5,
    i_sUser := GV.sUserLogged,
    i_sDescription := CONCAT(STR1 := 'Logged out: ', STR2 := GV.sUserLogged),
    iq_stParams := stDbParam,
    iq_bWrite := bWrite); // FB_WriteClick

// NETWORK 27
fbOperatorAction[2](
    i_bWrite := bOperatorAction[2],
    i_enEvent := 5,
    i_sUser := GV.sUserLogged,
    i_sDescription := 'Machine Power ON',
    iq_stParams := stDbParam,
    iq_bWrite := bWrite); // FB_WriteClick

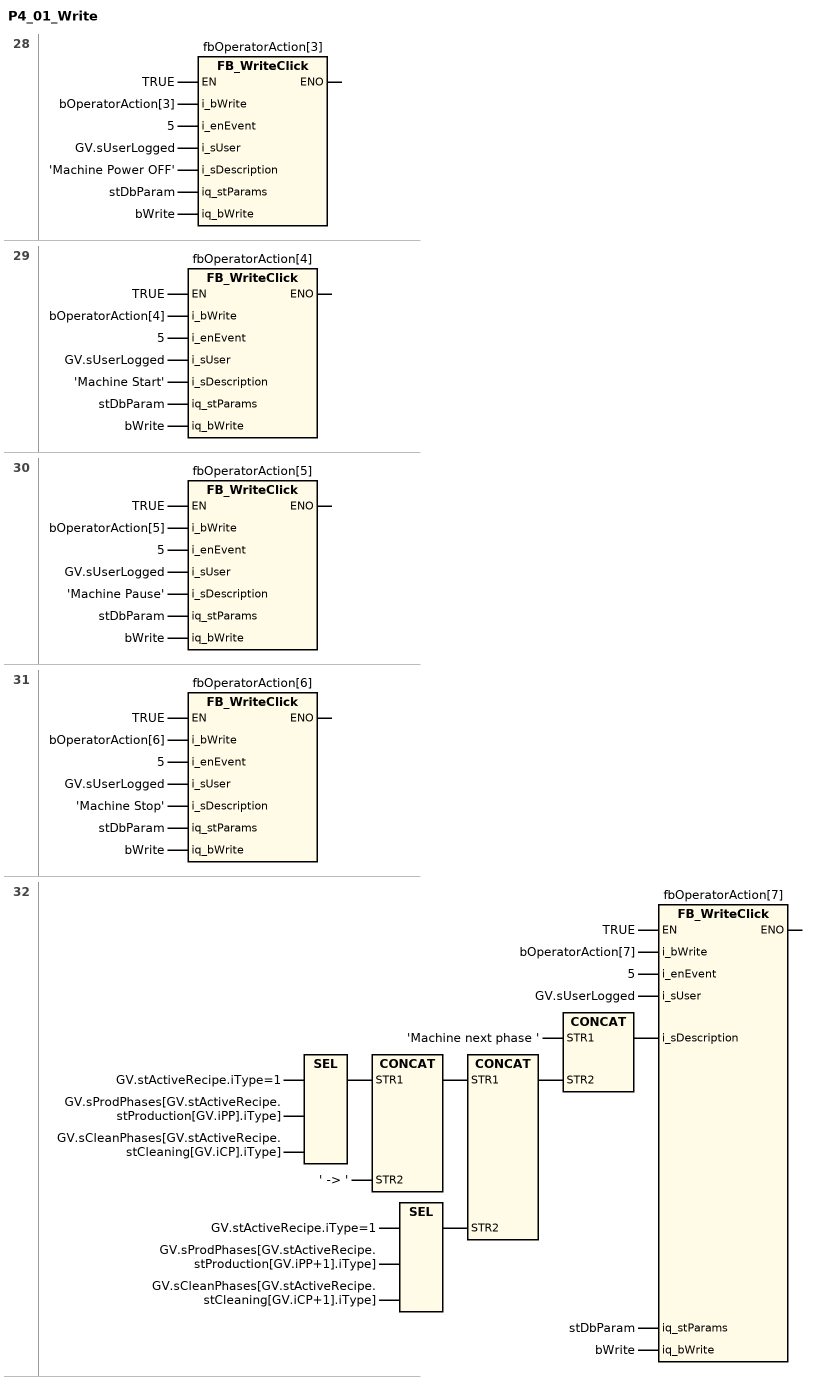
// NETWORK 28
fbOperatorAction[3](
    i_bWrite := bOperatorAction[3],
    i_enEvent := 5,
    i_sUser := GV.sUserLogged,
    i_sDescription := 'Machine Power OFF',
    iq_stParams := stDbParam,
    iq_bWrite := bWrite); // FB_WriteClick

// NETWORK 29
fbOperatorAction[4](
    i_bWrite := bOperatorAction[4],
    i_enEvent := 5,
    i_sUser := GV.sUserLogged,
    i_sDescription := 'Machine Start',
    iq_stParams := stDbParam,
    iq_bWrite := bWrite); // FB_WriteClick

// NETWORK 30
fbOperatorAction[5](
    i_bWrite := bOperatorAction[5],
    i_enEvent := 5,
    i_sUser := GV.sUserLogged,
    i_sDescription := 'Machine Pause',
    iq_stParams := stDbParam,
    iq_bWrite := bWrite); // FB_WriteClick

// NETWORK 31
fbOperatorAction[6](
    i_bWrite := bOperatorAction[6],
    i_enEvent := 5,
    i_sUser := GV.sUserLogged,
    i_sDescription := 'Machine Stop',
    iq_stParams := stDbParam,
    iq_bWrite := bWrite); // FB_WriteClick

// NETWORK 32
fbOperatorAction[7](
    i_bWrite := bOperatorAction[7],
    i_enEvent := 5,
    i_sUser := GV.sUserLogged,
    i_sDescription := CONCAT(STR1 := 'Machine next phase ', STR2 := CONCAT(STR1 := CONCAT(STR1 := SEL(GV.stActiveRecipe.iType=1, GV.sProdPhases[GV.stActiveRecipe.stProduction[GV.iPP].iType], GV.sCleanPhases[GV.stActiveRecipe.stCleaning[GV.iCP].iType]), STR2 := ' -> '), STR2 := SEL(GV.stActiveRecipe.iType=1, GV.sProdPhases[GV.stActiveRecipe.stProduction[GV.iPP+1].iType], GV.sCleanPhases[GV.stActiveRecipe.stCleaning[GV.iCP+1].iType]))),
    iq_stParams := stDbParam,
    iq_bWrite := bWrite); // FB_WriteClick

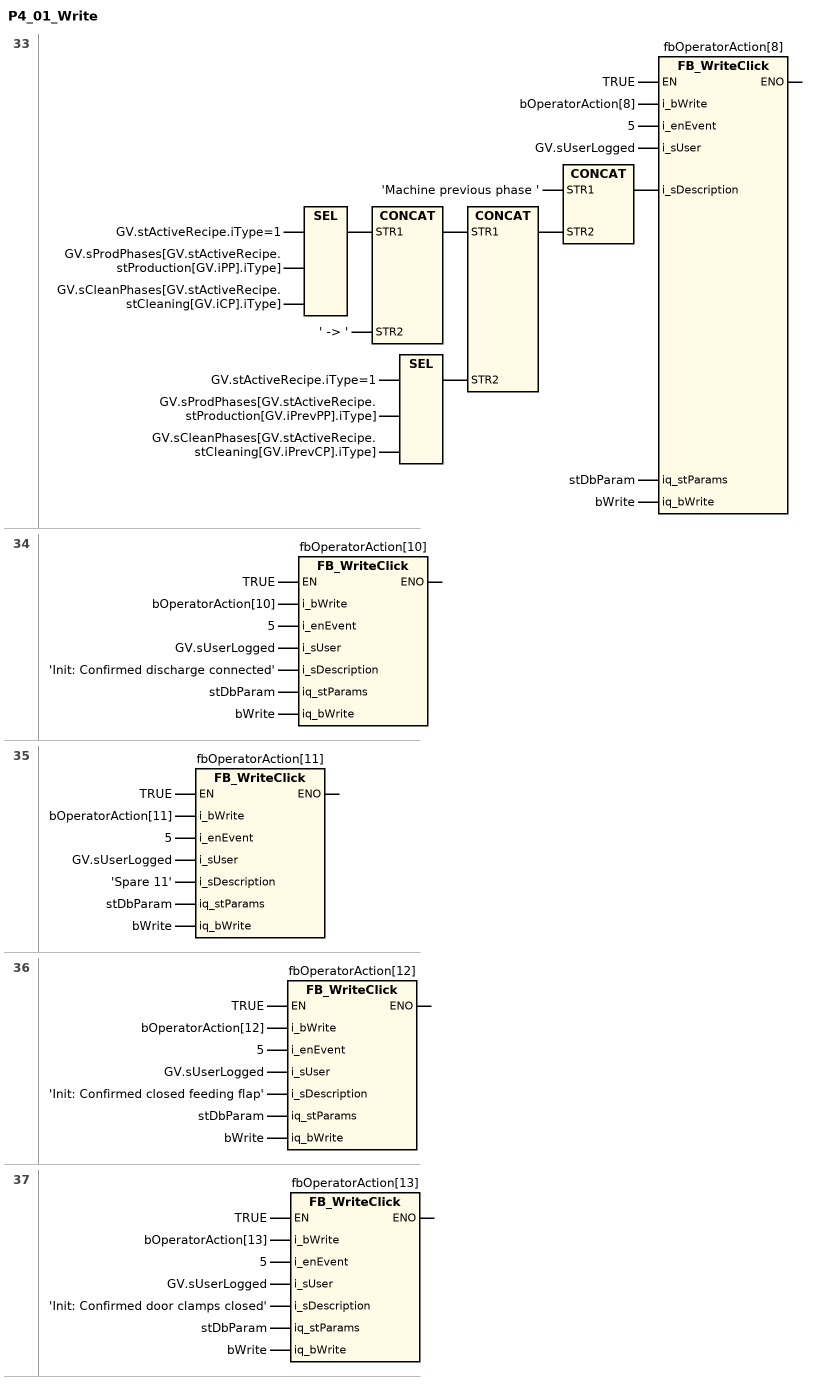
// NETWORK 33
fbOperatorAction[8](
    i_bWrite := bOperatorAction[8],
    i_enEvent := 5,
    i_sUser := GV.sUserLogged,
    i_sDescription := CONCAT(STR1 := 'Machine previous phase ', STR2 := CONCAT(STR1 := CONCAT(STR1 := SEL(GV.stActiveRecipe.iType=1, GV.sProdPhases[GV.stActiveRecipe.stProduction[GV.iPP].iType], GV.sCleanPhases[GV.stActiveRecipe.stCleaning[GV.iCP].iType]), STR2 := ' -> '), STR2 := SEL(GV.stActiveRecipe.iType=1, GV.sProdPhases[GV.stActiveRecipe.stProduction[GV.iPrevPP].iType], GV.sCleanPhases[GV.stActiveRecipe.stCleaning[GV.iPrevCP].iType]))),
    iq_stParams := stDbParam,
    iq_bWrite := bWrite); // FB_WriteClick

// NETWORK 34
fbOperatorAction[10](
    i_bWrite := bOperatorAction[10],
    i_enEvent := 5,
    i_sUser := GV.sUserLogged,
    i_sDescription := 'Init: Confirmed discharge connected',
    iq_stParams := stDbParam,
    iq_bWrite := bWrite); // FB_WriteClick

// NETWORK 35
fbOperatorAction[11](
    i_bWrite := bOperatorAction[11],
    i_enEvent := 5,
    i_sUser := GV.sUserLogged,
    i_sDescription := 'Spare 11',
    iq_stParams := stDbParam,
    iq_bWrite := bWrite); // FB_WriteClick

// NETWORK 36
fbOperatorAction[12](
    i_bWrite := bOperatorAction[12],
    i_enEvent := 5,
    i_sUser := GV.sUserLogged,
    i_sDescription := 'Init: Confirmed closed feeding flap',
    iq_stParams := stDbParam,
    iq_bWrite := bWrite); // FB_WriteClick

// NETWORK 37
fbOperatorAction[13](
    i_bWrite := bOperatorAction[13],
    i_enEvent := 5,
    i_sUser := GV.sUserLogged,
    i_sDescription := 'Init: Confirmed door clamps closed',
    iq_stParams := stDbParam,
    iq_bWrite := bWrite); // FB_WriteClick

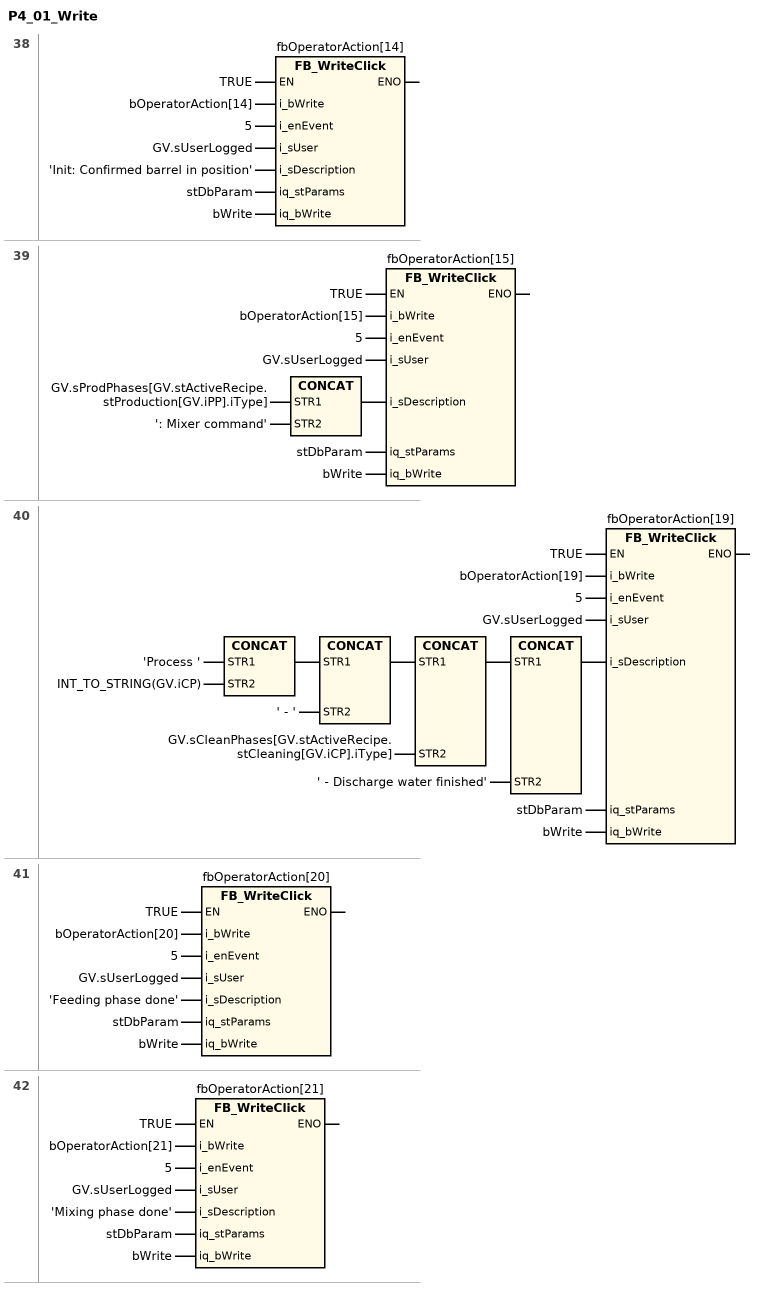
// NETWORK 38
fbOperatorAction[14](
    i_bWrite := bOperatorAction[14],
    i_enEvent := 5,
    i_sUser := GV.sUserLogged,
    i_sDescription := 'Init: Confirmed barrel in position',
    iq_stParams := stDbParam,
    iq_bWrite := bWrite); // FB_WriteClick

// NETWORK 39
fbOperatorAction[15](
    i_bWrite := bOperatorAction[15],
    i_enEvent := 5,
    i_sUser := GV.sUserLogged,
    i_sDescription := CONCAT(STR1 := GV.sProdPhases[GV.stActiveRecipe.stProduction[GV.iPP].iType], STR2 := ': Mixer command'),
    iq_stParams := stDbParam,
    iq_bWrite := bWrite); // FB_WriteClick

// NETWORK 40
fbOperatorAction[19](
    i_bWrite := bOperatorAction[19],
    i_enEvent := 5,
    i_sUser := GV.sUserLogged,
    i_sDescription := CONCAT(STR1 := CONCAT(STR1 := CONCAT(STR1 := CONCAT(STR1 := 'Process ', STR2 := INT_TO_STRING(GV.iCP)), STR2 := ' - '), STR2 := GV.sCleanPhases[GV.stActiveRecipe.stCleaning[GV.iCP].iType]), STR2 := ' - Discharge water finished'),
    iq_stParams := stDbParam,
    iq_bWrite := bWrite); // FB_WriteClick

// NETWORK 41
fbOperatorAction[20](
    i_bWrite := bOperatorAction[20],
    i_enEvent := 5,
    i_sUser := GV.sUserLogged,
    i_sDescription := 'Feeding phase done',
    iq_stParams := stDbParam,
    iq_bWrite := bWrite); // FB_WriteClick

// NETWORK 42
fbOperatorAction[21](
    i_bWrite := bOperatorAction[21],
    i_enEvent := 5,
    i_sUser := GV.sUserLogged,
    i_sDescription := 'Mixing phase done',
    iq_stParams := stDbParam,
    iq_bWrite := bWrite); // FB_WriteClick

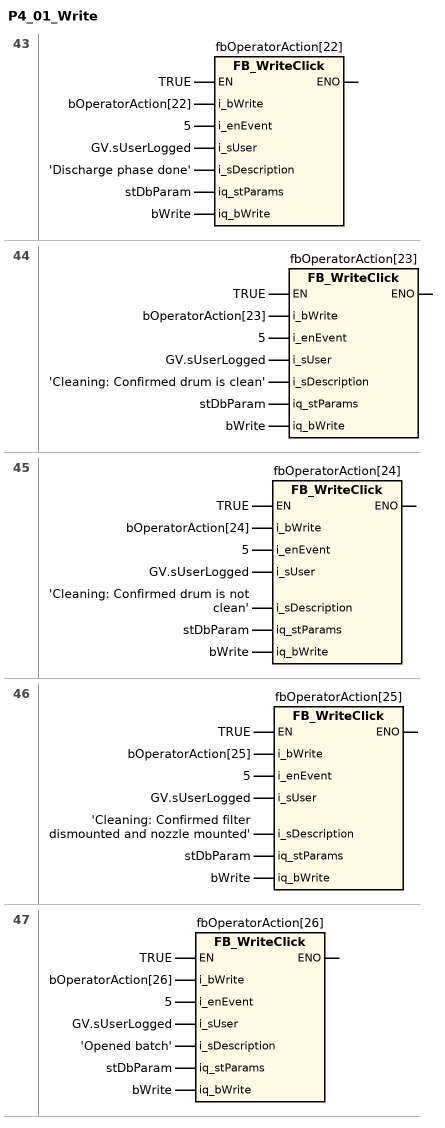
// NETWORK 43
fbOperatorAction[22](
    i_bWrite := bOperatorAction[22],
    i_enEvent := 5,
    i_sUser := GV.sUserLogged,
    i_sDescription := 'Discharge phase done',
    iq_stParams := stDbParam,
    iq_bWrite := bWrite); // FB_WriteClick

// NETWORK 44
fbOperatorAction[23](
    i_bWrite := bOperatorAction[23],
    i_enEvent := 5,
    i_sUser := GV.sUserLogged,
    i_sDescription := 'Cleaning: Confirmed drum is clean',
    iq_stParams := stDbParam,
    iq_bWrite := bWrite); // FB_WriteClick

// NETWORK 45
fbOperatorAction[24](
    i_bWrite := bOperatorAction[24],
    i_enEvent := 5,
    i_sUser := GV.sUserLogged,
    i_sDescription := 'Cleaning: Confirmed drum is not clean',
    iq_stParams := stDbParam,
    iq_bWrite := bWrite); // FB_WriteClick

// NETWORK 46
fbOperatorAction[25](
    i_bWrite := bOperatorAction[25],
    i_enEvent := 5,
    i_sUser := GV.sUserLogged,
    i_sDescription := 'Cleaning: Confirmed filter dismounted and nozzle mounted',
    iq_stParams := stDbParam,
    iq_bWrite := bWrite); // FB_WriteClick

// NETWORK 47
fbOperatorAction[26](
    i_bWrite := bOperatorAction[26],
    i_enEvent := 5,
    i_sUser := GV.sUserLogged,
    i_sDescription := 'Opened batch',
    iq_stParams := stDbParam,
    iq_bWrite := bWrite); // FB_WriteClick

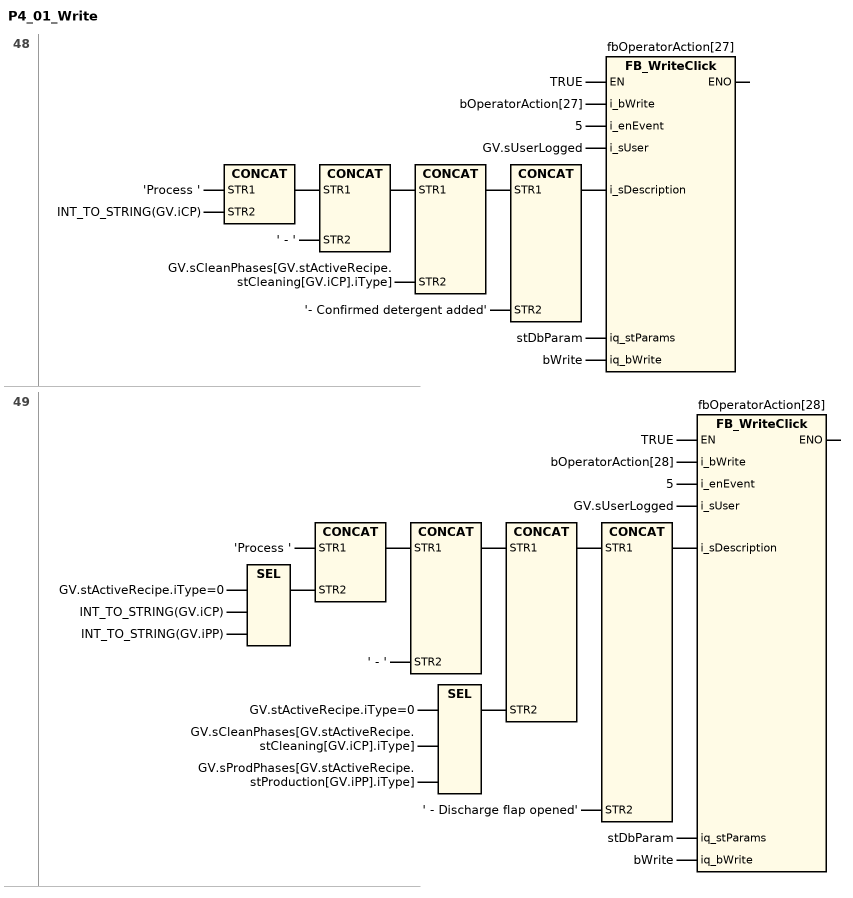
// NETWORK 48
fbOperatorAction[27](
    i_bWrite := bOperatorAction[27],
    i_enEvent := 5,
    i_sUser := GV.sUserLogged,
    i_sDescription := CONCAT(STR1 := CONCAT(STR1 := CONCAT(STR1 := CONCAT(STR1 := 'Process ', STR2 := INT_TO_STRING(GV.iCP)), STR2 := ' - '), STR2 := GV.sCleanPhases[GV.stActiveRecipe.stCleaning[GV.iCP].iType]), STR2 := '- Confirmed detergent added'),
    iq_stParams := stDbParam,
    iq_bWrite := bWrite); // FB_WriteClick

// NETWORK 49
fbOperatorAction[28](
    i_bWrite := bOperatorAction[28],
    i_enEvent := 5,
    i_sUser := GV.sUserLogged,
    i_sDescription := CONCAT(STR1 := CONCAT(STR1 := CONCAT(STR1 := CONCAT(STR1 := 'Process ', STR2 := SEL(GV.stActiveRecipe.iType=0, INT_TO_STRING(GV.iCP), INT_TO_STRING(GV.iPP))), STR2 := ' - '), STR2 := SEL(GV.stActiveRecipe.iType=0, GV.sCleanPhases[GV.stActiveRecipe.stCleaning[GV.iCP].iType], GV.sProdPhases[GV.stActiveRecipe.stProduction[GV.iPP].iType])), STR2 := ' - Discharge flap opened'),
    iq_stParams := stDbParam,
    iq_bWrite := bWrite); // FB_WriteClick

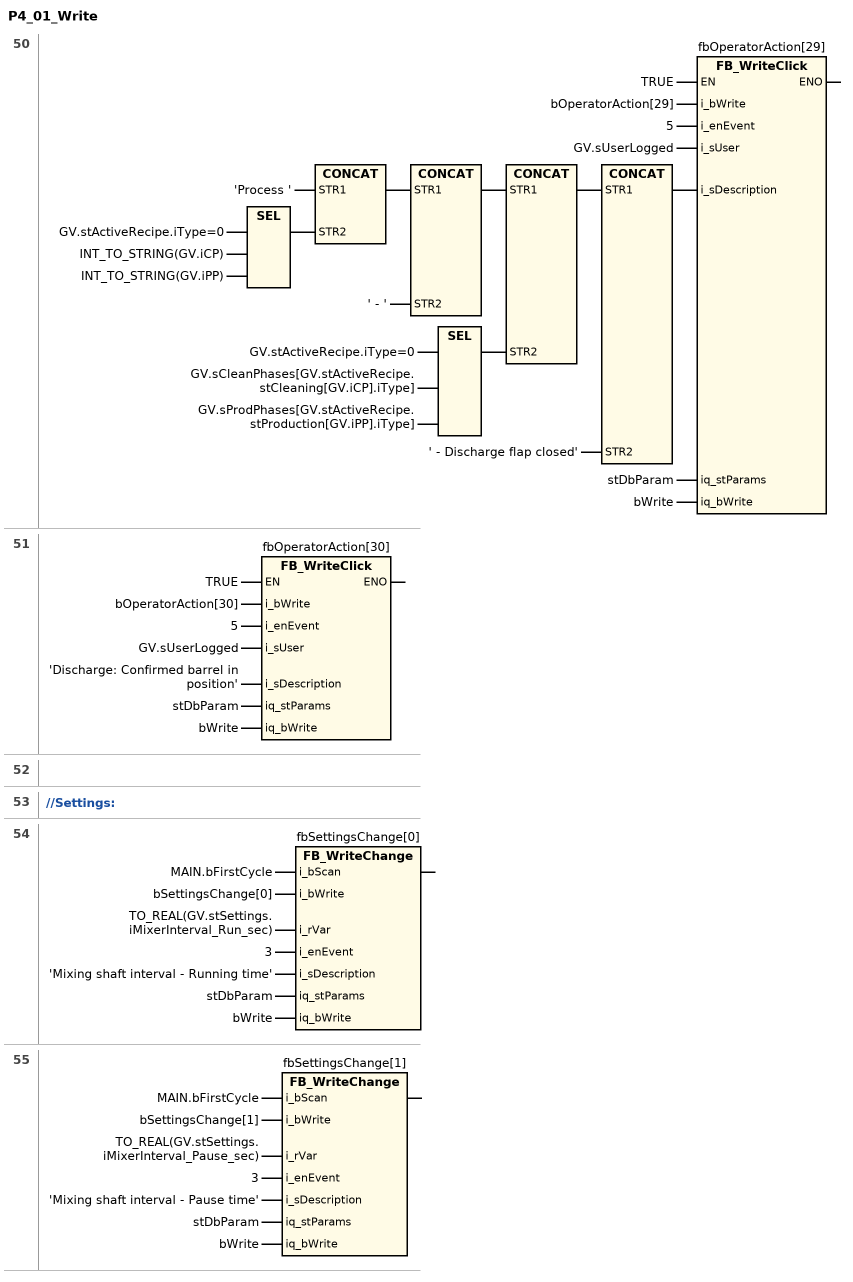
// NETWORK 50
fbOperatorAction[29](
    i_bWrite := bOperatorAction[29],
    i_enEvent := 5,
    i_sUser := GV.sUserLogged,
    i_sDescription := CONCAT(STR1 := CONCAT(STR1 := CONCAT(STR1 := CONCAT(STR1 := 'Process ', STR2 := SEL(GV.stActiveRecipe.iType=0, INT_TO_STRING(GV.iCP), INT_TO_STRING(GV.iPP))), STR2 := ' - '), STR2 := SEL(GV.stActiveRecipe.iType=0, GV.sCleanPhases[GV.stActiveRecipe.stCleaning[GV.iCP].iType], GV.sProdPhases[GV.stActiveRecipe.stProduction[GV.iPP].iType])), STR2 := ' - Discharge flap closed'),
    iq_stParams := stDbParam,
    iq_bWrite := bWrite); // FB_WriteClick

// NETWORK 51
fbOperatorAction[30](
    i_bWrite := bOperatorAction[30],
    i_enEvent := 5,
    i_sUser := GV.sUserLogged,
    i_sDescription := 'Discharge: Confirmed barrel in position',
    iq_stParams := stDbParam,
    iq_bWrite := bWrite); // FB_WriteClick

// NETWORK 52

// NETWORK 53
// label: //Settings

// NETWORK 54
fbSettingsChange[0](
    i_bScan := MAIN.bFirstCycle,
    i_bWrite := bSettingsChange[0],
    i_rVar := TO_REAL(GV.stSettings.iMixerInterval_Run_sec),
    i_enEvent := 3,
    i_sDescription := 'Mixing shaft interval - Running time',
    iq_stParams := stDbParam,
    iq_bWrite := bWrite); // FB_WriteChange

// NETWORK 55
fbSettingsChange[1](
    i_bScan := MAIN.bFirstCycle,
    i_bWrite := bSettingsChange[1],
    i_rVar := TO_REAL(GV.stSettings.iMixerInterval_Pause_sec),
    i_enEvent := 3,
    i_sDescription := 'Mixing shaft interval - Pause time',
    iq_stParams := stDbParam,
    iq_bWrite := bWrite); // FB_WriteChange

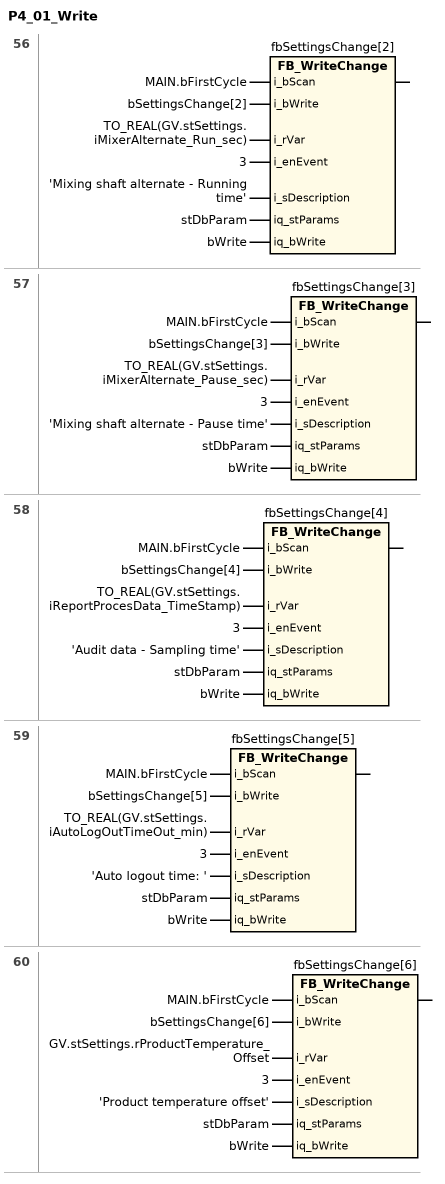
// NETWORK 56
fbSettingsChange[2](
    i_bScan := MAIN.bFirstCycle,
    i_bWrite := bSettingsChange[2],
    i_rVar := TO_REAL(GV.stSettings.iMixerAlternate_Run_sec),
    i_enEvent := 3,
    i_sDescription := 'Mixing shaft alternate - Running time',
    iq_stParams := stDbParam,
    iq_bWrite := bWrite); // FB_WriteChange

// NETWORK 57
fbSettingsChange[3](
    i_bScan := MAIN.bFirstCycle,
    i_bWrite := bSettingsChange[3],
    i_rVar := TO_REAL(GV.stSettings.iMixerAlternate_Pause_sec),
    i_enEvent := 3,
    i_sDescription := 'Mixing shaft alternate - Pause time',
    iq_stParams := stDbParam,
    iq_bWrite := bWrite); // FB_WriteChange

// NETWORK 58
fbSettingsChange[4](
    i_bScan := MAIN.bFirstCycle,
    i_bWrite := bSettingsChange[4],
    i_rVar := TO_REAL(GV.stSettings.iReportProcesData_TimeStamp),
    i_enEvent := 3,
    i_sDescription := 'Audit data - Sampling time',
    iq_stParams := stDbParam,
    iq_bWrite := bWrite); // FB_WriteChange

// NETWORK 59
fbSettingsChange[5](
    i_bScan := MAIN.bFirstCycle,
    i_bWrite := bSettingsChange[5],
    i_rVar := TO_REAL(GV.stSettings.iAutoLogOutTimeOut_min),
    i_enEvent := 3,
    i_sDescription := 'Auto logout time: ',
    iq_stParams := stDbParam,
    iq_bWrite := bWrite); // FB_WriteChange

// NETWORK 60
fbSettingsChange[6](
    i_bScan := MAIN.bFirstCycle,
    i_bWrite := bSettingsChange[6],
    i_rVar := GV.stSettings.rProductTemperature_Offset,
    i_enEvent := 3,
    i_sDescription := 'Product temperature offset',
    iq_stParams := stDbParam,
    iq_bWrite := bWrite); // FB_WriteChange

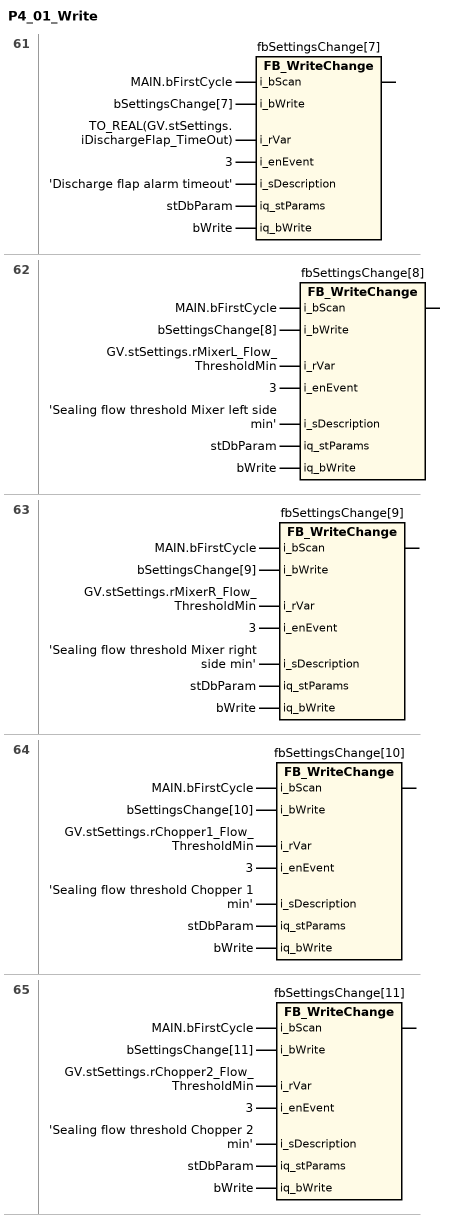
// NETWORK 61
fbSettingsChange[7](
    i_bScan := MAIN.bFirstCycle,
    i_bWrite := bSettingsChange[7],
    i_rVar := TO_REAL(GV.stSettings.iDischargeFlap_TimeOut),
    i_enEvent := 3,
    i_sDescription := 'Discharge flap alarm timeout',
    iq_stParams := stDbParam,
    iq_bWrite := bWrite); // FB_WriteChange

// NETWORK 62
fbSettingsChange[8](
    i_bScan := MAIN.bFirstCycle,
    i_bWrite := bSettingsChange[8],
    i_rVar := GV.stSettings.rMixerL_Flow_ThresholdMin,
    i_enEvent := 3,
    i_sDescription := 'Sealing flow threshold Mixer left side min',
    iq_stParams := stDbParam,
    iq_bWrite := bWrite); // FB_WriteChange

// NETWORK 63
fbSettingsChange[9](
    i_bScan := MAIN.bFirstCycle,
    i_bWrite := bSettingsChange[9],
    i_rVar := GV.stSettings.rMixerR_Flow_ThresholdMin,
    i_enEvent := 3,
    i_sDescription := 'Sealing flow threshold Mixer right side min',
    iq_stParams := stDbParam,
    iq_bWrite := bWrite); // FB_WriteChange

// NETWORK 64
fbSettingsChange[10](
    i_bScan := MAIN.bFirstCycle,
    i_bWrite := bSettingsChange[10],
    i_rVar := GV.stSettings.rChopper1_Flow_ThresholdMin,
    i_enEvent := 3,
    i_sDescription := 'Sealing flow threshold Chopper 1 min',
    iq_stParams := stDbParam,
    iq_bWrite := bWrite); // FB_WriteChange

// NETWORK 65
fbSettingsChange[11](
    i_bScan := MAIN.bFirstCycle,
    i_bWrite := bSettingsChange[11],
    i_rVar := GV.stSettings.rChopper2_Flow_ThresholdMin,
    i_enEvent := 3,
    i_sDescription := 'Sealing flow threshold Chopper 2 min',
    iq_stParams := stDbParam,
    iq_bWrite := bWrite); // FB_WriteChange

